REGION Network 8: SALIDAS - Baliza ROJA
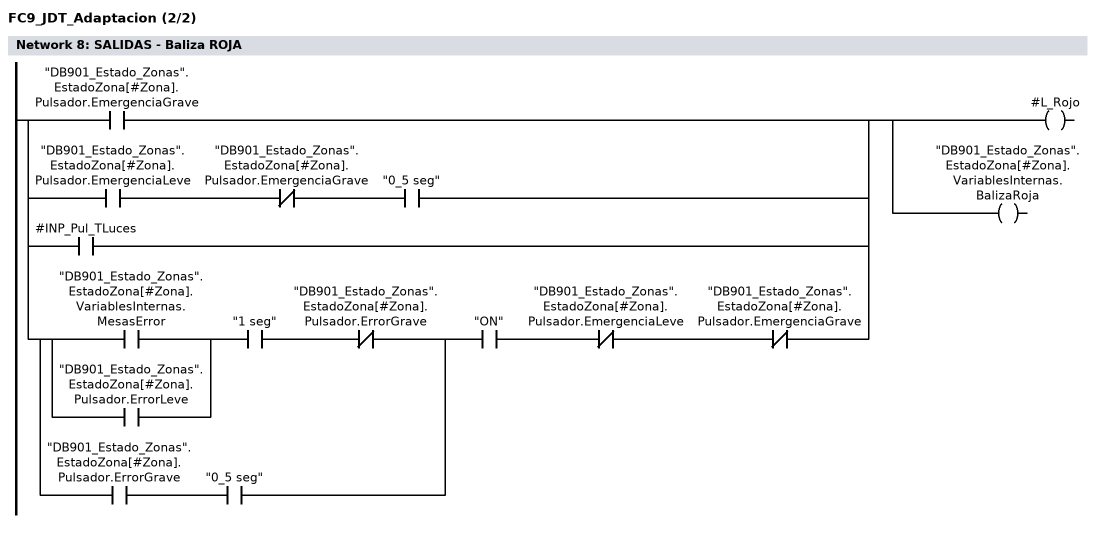
   RUNG wire#powerrail
      Contact( "DB901_Estado_Zonas".EstadoZona[#Zona].Pulsador.EmergenciaGrave )
      wire#w1
      Coil( #L_Rojo )
   END_RUNG
   RUNG wire#powerrail
      Contact( "DB901_Estado_Zonas".EstadoZona[#Zona].Pulsador.EmergenciaLeve )
      I_Contact( "DB901_Estado_Zonas".EstadoZona[#Zona].Pulsador.EmergenciaGrave )
      Contact( "0_5 seg" )
   END_RUNG wire#w1
   RUNG wire#powerrail
      Contact( #INP_Pul_TLuces )
   END_RUNG wire#w1
   RUNG wire#powerrail
      Contact( "DB901_Estado_Zonas".EstadoZona[#Zona].VariablesInternas.MesasError )
      wire#w2
      Contact( "1 seg" )
      I_Contact( "DB901_Estado_Zonas".EstadoZona[#Zona].Pulsador.ErrorGrave )
      wire#w3
      Contact( "ON" )
      I_Contact( "DB901_Estado_Zonas".EstadoZona[#Zona].Pulsador.EmergenciaLeve )
      I_Contact( "DB901_Estado_Zonas".EstadoZona[#Zona].Pulsador.EmergenciaGrave )
   END_RUNG wire#w1
   RUNG wire#powerrail
      Contact( "DB901_Estado_Zonas".EstadoZona[#Zona].Pulsador.ErrorLeve )
   END_RUNG wire#w2
   RUNG wire#powerrail
      Contact( "DB901_Estado_Zonas".EstadoZona[#Zona].Pulsador.ErrorGrave )
      Contact( "0_5 seg" )
   END_RUNG wire#w3
   RUNG wire#w1
      Coil( "DB901_Estado_Zonas".EstadoZona[#Zona].VariablesInternas.BalizaRoja )
   END_RUNG
   // the same network as SCL:
   #L_Rojo := "DB901_Estado_Zonas".EstadoZona[#Zona].Pulsador.EmergenciaGrave OR ("DB901_Estado_Zonas".EstadoZona[#Zona].Pulsador.EmergenciaLeve AND NOT "DB901_Estado_Zonas".EstadoZona[#Zona].Pulsador.EmergenciaGrave AND "0_5 seg") OR #INP_Pul_TLuces OR (((("DB901_Estado_Zonas".EstadoZona[#Zona].VariablesInternas.MesasError OR "DB901_Estado_Zonas".EstadoZona[#Zona].Pulsador.ErrorLeve) AND "1 seg" AND NOT "DB901_Estado_Zonas".EstadoZona[#Zona].Pulsador.ErrorGrave) OR ("DB901_Estado_Zonas".EstadoZona[#Zona].Pulsador.ErrorGrave AND "0_5 seg")) AND "ON" AND NOT "DB901_Estado_Zonas".EstadoZona[#Zona].Pulsador.EmergenciaLeve AND NOT "DB901_Estado_Zonas".EstadoZona[#Zona].Pulsador.EmergenciaGrave);
   "DB901_Estado_Zonas".EstadoZona[#Zona].VariablesInternas.BalizaRoja := #L_Rojo;
END_REGION
END_FUNCTION

FUNCTION_BLOCK "FB600_ControlPosicion_Quimarox"   // FB600, LAD
{ S7_Optimized_Access := 'FALSE' }
AUTHOR : Naibes
// stored: AutoNumber false, SetENOAutomatically false
   VAR_INPUT
      ID_Quimarox : UInt;
      Detector_paso_cero : Bool;
      V_Cnt_Tout_paso_Cero : UDInt;
      Dato_encoder : DInt;   // Tiene que ser una entrada del DB de encoders
   END_VAR
   VAR_OUTPUT
      numero_vagon_entrada : Int;
      avance_vagon_entrada : Int;
      avance_total : Int;
   END_VAR
   VAR
      maux_fp_detect_cero : Bool;
      mem_cnt_tout : UDInt;
      total_registros : Int;
   END_VAR
   VAR_TEMP
      contador_elementos : Int;
      pulsos_transcurridos : DInt;
      avance_vagon_ref : DInt;
      num_vag_in : Int;
      Avance_vag_inic : Int;
      aux_int : Int;
      Avance_vagon_X : Int;
      salto : Int;
      basura : Bool;
   END_VAR
BEGIN

NETWORK
TITLE = Variable provisional
//=====================================================================================================================

//=====================================================================================================================

NETWORK
TITLE = 
// Control de posicionamiento y memorias de encoder

      CALL  "FC600_ini+ref_dato_encoder_NEW"
      ( Detector_referencia := #Detector_paso_cero,
        ID_Quimarox         := #ID_Quimarox,
        dato_encoder_actual := #Dato_encoder,
        V_cnt_tout_refresco := #V_Cnt_Tout_paso_Cero,
        m_aux_pf_detect     := #maux_fp_detect_cero,
        MEM_CNT_TOUT        := #mem_cnt_tout
      );


NETWORK
TITLE = Variable provisional
      SET;
      A     "DB600_ConfigQuimarox".Quimarox[#ID_Quimarox].datos_config.DatosTrabajo.Error_Referenciacion;  // #Error_Referenciacion
      R     "DB600_ConfigQuimarox".Quimarox[#ID_Quimarox].datos_config.DatosTrabajo.Memoria_Inicializacion;  //#Mem_Inicializacion

NETWORK
TITLE = Borrado de DB Posiciones asociadas a elementos
// aqui se borran todas las posiciones asociadas a los elementos para luego 
// posteriormente cargar los datos que correspondan. Esto lo hacemos antes de 
// comprobar si está inicializado o no para que si perdemos la referencia dejemos 
// de tener datos.
//=====================================================================================================================

      L     1;  //Iniciamos Cont. Bytes a Borrar     Cuidado con los temporales, inicializar siempre
      T     #contador_elementos;


bucl: NOP   0;
//=====================================================================================================================
//limpia los datos antes de calcular los nuevos

      SET;
      R     "DB602_ElementosQuimarox".Quimarox[#ID_Quimarox].Elementos[#contador_elementos].Hay_Carrier_en_ventana;  //Vagon_en_Ventana
      L     0;
      T     "DB602_ElementosQuimarox".Quimarox[#ID_Quimarox].Elementos[#contador_elementos].Numero_carrier;  //Vagon_Asociado
      T     "DB602_ElementosQuimarox".Quimarox[#ID_Quimarox].Elementos[#contador_elementos].Avance_carrier;  //Posicion_Vagon


      L     #contador_elementos;
      L     "CTE_MaxNumElementos";
      >=I;
      JC    cont;

      L     1;
      L     #contador_elementos;
      +I;
      T     #contador_elementos;

      JU    bucl;
//=====================================================================================================================

NETWORK
TITLE = 
//=====================================================================================================================

cont: AN    "DB600_ConfigQuimarox".Quimarox[#ID_Quimarox].datos_config.DatosTrabajo.Memoria_Inicializacion;
      JC    fin1;  //el primer vagon y no podemos calcular nada

//=====================================================================================================================

NETWORK
TITLE = 
// con el dato del encoder de referencia del primer vagon calculamos el elemento 
// que se encuentra en la entrada del sorter para utilizarlo de vagon de referencia
//===================================================================================================
//aqui comprobaremos si ha pasado por el máximo o no y en funcion de eso calcularemos el numero
//de pulsos que han transcurrido desde la referenciación del primer vagon
//====================================================================================================

      L     "DB600_ConfigQuimarox".Quimarox[#ID_Quimarox].datos_config.DatosTrabajo.Memoria_Dato_Encoder;  //#Mem_Dato_Encoder
      L     #Dato_encoder;
      >D;
      JCN   MEN;

      L     "DB600_ConfigQuimarox".Quimarox[#ID_Quimarox].datos_config.maximo_encoder;
      L     "DB600_ConfigQuimarox".Quimarox[#ID_Quimarox].datos_config.DatosTrabajo.Memoria_Dato_Encoder;
      -D;
      L     #Dato_encoder;
      +D;
      T     #pulsos_transcurridos;
      JU    CLC;

//=====================================================================================================================

MEN:  L     #Dato_encoder;
      L     "DB600_ConfigQuimarox".Quimarox[#ID_Quimarox].datos_config.DatosTrabajo.Memoria_Dato_Encoder;
      -D;
      T     #pulsos_transcurridos;


//============================================================================================================================================
// NIEVES: Calculo del avance del vagón de referencia

CLC:  L     #pulsos_transcurridos;
      DTR;
      L     "DB600_ConfigQuimarox".Quimarox[#ID_Quimarox].datos_config.relacion_mm_pulso;  // #Datos_config.relacion_mm_pulso
      *R;
      RND+;
      L     "DB600_ConfigQuimarox".Quimarox[#ID_Quimarox].datos_config.dist_ini_vag_a_phs_mm;  //distancia del punto de deteccion de referencia al punto de referencia 0
      ITD;
      +D;
      T     #avance_vagon_ref;  //en mm

//=====================================================================================================================

//con el dato del avance del vagon de referencia calculamos cual es el vagon que esta en el inicio del sorter
//y cuando ha avanzado respecto del punto de referencia para con este dato calcular la posicion del resto


NETWORK
TITLE = Calculo de posicón del primer vagón
// en funcion del avance del primer vagon calculamos cual es el vagon que se 
// encuentra en el inicio del sorter y cuanto ha avanzado desde el punto de 
// referencia
//=====================================================================================================================
//si no hace bien lo del numero de vagon revisar este punto
      L     #avance_vagon_ref;
      L     "DB600_ConfigQuimarox".Quimarox[#ID_Quimarox].datos_config.Long_Vagon_mm;
      ITD;
      /D;
      L     1;
      +D;
      DTB;
      BTI;
      T     #num_vag_in;  //Calcula y guarda Vagon en posición inicial

      L     #num_vag_in;
      L     "DB600_ConfigQuimarox".Quimarox[#ID_Quimarox].datos_config.Numero_vagones;

      <=I;
      JC    p_1;

//=====================================================================================================================

      L     #num_vag_in;
      L     "DB600_ConfigQuimarox".Quimarox[#ID_Quimarox].datos_config.Numero_vagones;
      -I;
      T     #numero_vagon_entrada;
      JU    p_2;

//=====================================================================================================================
p_1:  L     #num_vag_in;
      T     #numero_vagon_entrada;

//=====================================================================================================================
p_2:  L     #avance_vagon_ref;
      L     "DB600_ConfigQuimarox".Quimarox[#ID_Quimarox].datos_config.Long_Vagon_mm;
      MOD;
      T     #avance_vagon_entrada;
      T     #Avance_vag_inic;  //Calcula y guarda avance Vagon actual en posición inicial

      L     #pulsos_transcurridos;  // Calcula el avance total desde origen
      DTR;
      L     "DB600_ConfigQuimarox".Quimarox[#ID_Quimarox].datos_config.relacion_mm_pulso;
      *R;
      RND+;
      T     #avance_total;

//=====================================================================================================================

NETWORK
TITLE = calculo posicon vagon todos elementos
// aqui vamos realizando los saltos a cada uno de los elementos, calculamos lo que 
// ha avanzado el vagon y si entra dentro de los limites establecidos para dicho 
// elemento cargamos el numero de vagon correspondiente en la posicion asociada a 
// dicho elemento
//===================================================================================================================================

      L     1;
      T     #contador_elementos;

//=====================================================================================================================
//aqui el calculo de lo que ha avanzado el vagon para dicho elemento
//NIEVES


sige: NOP   0;

//=====================================================================================================================

      L     "DB602_ElementosQuimarox".Quimarox[#ID_Quimarox].Elementos[#contador_elementos].posicion_real_elemento;  //#datos_elemento_actual.posicion_real_elemento
      TRUNC;
      L     "DB600_ConfigQuimarox".Quimarox[#ID_Quimarox].datos_config.Long_Vagon_mm;
      ITD;
      MOD;
      T     #aux_int;
      L     "DB600_ConfigQuimarox".Quimarox[#ID_Quimarox].datos_config.Long_Vagon_mm;
      L     #aux_int;
      -I;  //Avance del vagon para el elemento tratado
      L     #Avance_vag_inic;
      +I;
      L     "DB600_ConfigQuimarox".Quimarox[#ID_Quimarox].datos_config.Long_Vagon_mm;
      MOD;
      T     #Avance_vagon_X;

//=====================================================================================================================

NETWORK
TITLE = comparación de la ventana del elemento segun grado de avance
// aqui la comparacion primero con el rango inferior y luego con el rango superior
//=====================================================================================================================
      CLR;
      =     "DB602_ElementosQuimarox".Quimarox[#ID_Quimarox].Elementos[#contador_elementos].Hay_Carrier_en_ventana;  //Inicio Validación elemento en rango Ventana


      L     "DB602_ElementosQuimarox".Quimarox[#ID_Quimarox].Elementos[#contador_elementos].ventana_minima;
      L     #Avance_vagon_X;
      >I;
      JC    vent;

//=====================================================================================================================

      L     "DB602_ElementosQuimarox".Quimarox[#ID_Quimarox].Elementos[#contador_elementos].ventana_maxima;  //apunta a la posicion maxima
      L     #Avance_vagon_X;
      <I;
      JC    vent;

      SET;
      =     "DB602_ElementosQuimarox".Quimarox[#ID_Quimarox].Elementos[#contador_elementos].Hay_Carrier_en_ventana;

//=====================================================================================================================




NETWORK
TITLE = calcular el número de vagón que corresponde
// aqui si se cumple que esta entre los dos rangos, calculamos el numero de vagon 
// que corresponde y lo cargamos en la correspondiente posicion asociada
// 
// al finalizar comprobar que no estamos en el ultimo elemento, si lo estamos, 
// saltar al final, y si no lo estamos pasa al siguiente elemento y spa sige
//=====================================================================================================================
//aqui calculamos el vagon que esta en frente del elemento
// para poder hacer el redondeo tenemos que hacer todo el cálculo en real

vent: L     "DB602_ElementosQuimarox".Quimarox[#ID_Quimarox].Elementos[#contador_elementos].posicion_real_elemento;
      L     #Avance_vag_inic;
      ITD;
      DTR;
      -R;
      L     "DB600_ConfigQuimarox".Quimarox[#ID_Quimarox].datos_config.Long_Vagon_mm;
      ITD;
      DTR;
      /R;
      RND+;
      T     #salto;
      L     #num_vag_in;
      L     #salto;
      -I;
      T     #aux_int;

      L     #aux_int;
      L     1;
      <I;
      JCN   p_3;


//=====================================================================================================================
      L     #aux_int;
      L     "DB600_ConfigQuimarox".Quimarox[#ID_Quimarox].datos_config.Numero_vagones;
      +I;
      T     #aux_int;


//=====================================================================================================================
p_3:  L     #aux_int;
      L     "DB600_ConfigQuimarox".Quimarox[#ID_Quimarox].datos_config.Numero_vagones;
      >I;
      JCN   carg;

      L     #aux_int;
      L     "DB600_ConfigQuimarox".Quimarox[#ID_Quimarox].datos_config.Numero_vagones;
      -I;
      T     #aux_int;

//=====================================================================================================================
carg: L     #aux_int;
      T     "DB602_ElementosQuimarox".Quimarox[#ID_Quimarox].Elementos[#contador_elementos].Numero_carrier;

      L     #Avance_vagon_X;
      T     "DB602_ElementosQuimarox".Quimarox[#ID_Quimarox].Elementos[#contador_elementos].Avance_carrier;

//=====================================================================================================================

      L     #contador_elementos;
      L     "CTE_MaxNumElementos";
      ==I;
      JC    fin;

      L     #contador_elementos;
      L     1;
      +I;
      T     #contador_elementos;

      JU    sige;

//=====================================================================================================================

NETWORK
TITLE = 
//=====================================================================================================================
fin:  BE;


//=====================================================================================================================
fin1: L     0;
      T     #numero_vagon_entrada;
      T     #avance_vagon_entrada;


//=====================================================================================================================
END_FUNCTION_BLOCK

FUNCTION_BLOCK "FB607_SalidaMovil_Frontal_Quimarox"   // FB607, LAD
{ S7_Optimized_Access := 'FALSE' }
// stored: AutoNumber false, SetENOAutomatically false
   VAR_INPUT
      MesaDeDescarga : UInt;
      ID_Quimarox : UInt;
      ID_Elemento : UInt;
      DestinoAsociado : UInt;
      pHs_PosicionDescarga : Bool;
      pHs_Protrusion : Bool;
      En_PosicionReposo : Bool;
      Corte_PosicionReposo : Bool;
      Corte_PosicionDesCarga : Bool;
      En_PosicionDescarga : Bool;
      Permiso_DeDesCarga : Bool;
      V_Filtro_pHsPresencia : Int;
      Pto_Ajuste_1 : Int;   // en mm (paso a lenta en posicionamiento a descarga de transportador)
      Pto_Ajuste_2 : Int;   // en mm (timeout movimiento posicion descarga del transportador)
      Pto_Ajuste_3 : Int;   // en mm (paso a lenta en posicionamiento reposo del transportador)
      Pto_Ajuste_4 : Int;   // en mm (timeout movimiento posicion reposo del transportador)
   END_VAR
   VAR_OUTPUT
      NXT_DescargaActiva : Bool;
      ElevadorEnLenta : Bool;
      PararElevador : Bool;
      Ir_PosicionReposo : Bool;
      Ir_PosicionDescarga : Bool;
   END_VAR
   VAR
      FILTRO_pHsPresencia : "FB910_CNT_UHS";
      EstadoAsociadoEnMesa : UInt;
      Ultimo_PeineTratado : UInt;
      Aux_PeineEnDesCarga { ExternalAccessible := 'False'; ExternalVisible := 'False'; ExternalWritable := 'False'} : UInt;
   END_VAR
   VAR_TEMP
      MesaQuimarox : UInt;
      NumeroUT : UInt;
      Vagon_Siguiente : Int;
      EsMesaTL : Bool;
      FILTRO_PosicionDesCarga : Bool;
   END_VAR
BEGIN

NETWORK
TITLE = ERROR - Rearme
/////////////////////////////////////////////////////////////
/////////////////////////////////////////////////////////////
/////////////////////////////////////////////////////////////
// Rearne de Errores
      SET;
      A     "DB902_Estado_ZonaMesa".EstadoMesas[#MesaDeDescarga].Rearme_CBx;
      O     "DB902_Estado_ZonaMesa".EstadoMesas[#MesaDeDescarga].PerReset_CBx;
      R     "DB900_Estado_Mesas".EstadoVI[#MesaDeDescarga].Error_Mx;
      R     "DB900_Estado_Mesas".EstadoVI[#MesaDeDescarga].Err_Protusion;
      R     "DB900_Estado_Mesas".EstadoVI[#MesaDeDescarga].Err_TOut_Avance_E1_E3;
      R     "DB900_Estado_Mesas".EstadoVI[#MesaDeDescarga].Err_Tout_Sacar;
      R     "DB900_Estado_Mesas".EstadoVI[#MesaDeDescarga].Err_Tout_Recoger;

      R     "DB900_Estado_Mesas".EstadoVI[#MesaDeDescarga].Err_DatosPLC;



NETWORK
TITLE = HMI - Entradas y Salidas de la Mesa
/////////////////////////////////////////////////////////////
/////////////////////////////////////////////////////////////
/////////////////////////////////////////////////////////////
// Entradas
      SET;
      A     #pHs_PosicionDescarga;
      =     "DB904_Estado_Maquinas".EstadoVI[#MesaDeDescarga].Byte7_bit4;
      SET;
      A     #pHs_Protrusion;
      =     "DB904_Estado_Maquinas".EstadoVI[#MesaDeDescarga].Byte9_bit0;

      SET;
      A     #En_PosicionReposo;
      =     "DB904_Estado_Maquinas".EstadoVI[#MesaDeDescarga].Byte8_bit4;
      SET;
      A     #Corte_PosicionReposo;
      =     "DB904_Estado_Maquinas".EstadoVI[#MesaDeDescarga].Byte7_bit6;
      SET;
      A     #Corte_PosicionDesCarga;
      =     "DB904_Estado_Maquinas".EstadoVI[#MesaDeDescarga].Byte7_bit7;
      SET;
      A     #En_PosicionDescarga;
      =     "DB904_Estado_Maquinas".EstadoVI[#MesaDeDescarga].Byte8_bit5;


// Salidas
      SET;
      A     #NXT_DescargaActiva;
      =     "DB900_Estado_Mesas".EstadoVI[#MesaDeDescarga].Sa_Giro_180;
      SET;
      A     #Ir_PosicionReposo;
      =     "DB900_Estado_Mesas".EstadoVI[#MesaDeDescarga].Sa_Trans_Baj;
      SET;
      A     #Ir_PosicionDescarga;
      =     "DB900_Estado_Mesas".EstadoVI[#MesaDeDescarga].Sa_Trans_Sub;



NETWORK
TITLE = Comprobacion de que la MESA es de TRACKING
/////////////////////////////////////////////////////////////////////////////////////
/////////////////////////////////////////////////////////////////////////////////////
/////////////////////////////////////////////////////////////////////////////////////
// Comprobar si es una Mesa de Tracking o Routing
      SET;
      A     "DB850_DefinicionMesas".Mesa[#MesaDeDescarga].ConfigMesa.MesaTL;
      =     #EsMesaTL;



NETWORK
TITLE = Inicializacio PREVIA
/////////////////////////////////////////////////////////////////////////////////////
/////////////////////////////////////////////////////////////////////////////////////
/////////////////////////////////////////////////////////////////////////////////////
      CLR;
      =     #ElevadorEnLenta;
      =     #PararElevador;

      CLR;
      =     #NXT_DescargaActiva;

      CLR;
      =     #Ir_PosicionReposo;
      =     #Ir_PosicionDescarga;



NETWORK
TITLE = SISTEMA - Reset
/////////////////////////////////////////////////////////////
/////////////////////////////////////////////////////////////
/////////////////////////////////////////////////////////////
// - Existe RESET ??
      SET;
      AN    "DB902_Estado_ZonaMesa".EstadoMesas[#MesaDeDescarga].PerReset_CBx;  //#Estado_CBx.PerReset_CBx
      JC    NoRealizandose_Reset;

      L     0;
      T     #EstadoAsociadoEnMesa;
      T     #Ultimo_PeineTratado;


/////////////////////////////////////////////////////////////
/////////////////////////////////////////////////////////////
/////////////////////////////////////////////////////////////
// - Final Tratamiento del RESET
NoRealizandose_Reset:NOP   0;



NETWORK
TITLE = >>>>>>>>>>>>>>>>>>>>>>>>>>>>>>>>>>>>>>>>>>>>>>>>>>>>>>>>>>>>>>>>>>>

REGION Network 7: FILTRO - pHs de Presencia
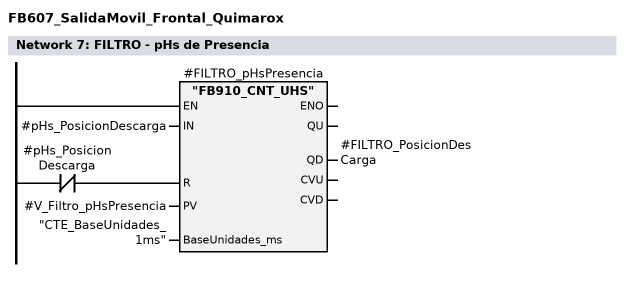
   RUNG wire#powerrail
      #FILTRO_pHsPresencia(R := wire#w1, IN := #pHs_PosicionDescarga, PV := #V_Filtro_pHsPresencia, BaseUnidades_ms := "CTE_BaseUnidades_1ms", QU =>, QD => #FILTRO_PosicionDesCarga, CVU =>, CVD =>)
   END_RUNG
   RUNG wire#powerrail
      I_Contact( #pHs_PosicionDescarga )
   END_RUNG wire#w1
   // the same network as SCL:
   #FILTRO_pHsPresencia(IN := #pHs_PosicionDescarga,   // "FB910_CNT_UHS"
                        R := NOT #pHs_PosicionDescarga,
                        PV := #V_Filtro_pHsPresencia,
                        BaseUnidades_ms := "CTE_BaseUnidades_1ms",
                        QD => #FILTRO_PosicionDesCarga);
END_REGION

NETWORK
TITLE = >>>>>>>>>>>>>>>>>>>>>>>>>>>>>>>>>>>>>>>>>>>>>>>>>>>>>>>>>>>>>>>>>>>

NETWORK
TITLE = Control Etapa activa >>> DISTRIBUCION
/////////////////////////////////////////////////////////////////////////////////////
/////////////////////////////////////////////////////////////////////////////////////
/////////////////////////////////////////////////////////////////////////////////////
// listado de saltos de programa
      L     #EstadoAsociadoEnMesa;

      JL    ETAPA_PorDefecto;
      JU    ETAPA_00_EnReset;
      JU    ETAPA_01_EnReposo;

      JU    ETAPA_02_EsperaPermisoDeDescarga;
      JU    ETAPA_03_MoverPosicionDescarga;
      JU    ETAPA_04_PreparadoParaDescarga;
      JU    ETAPA_05_FinDescarga;
      JU    ETAPA_06_MoverPosicionReposo;

      JU    ETAPA_PorDefecto;
      JU    ETAPA_PorDefecto;
      JU    ETAPA_PorDefecto;

      JU    ETAPA_10_ResetVacio_EsperaDesCargaDePeine;
      JU    ETAPA_11_ResetVacio_RecogerCargaDePeine;
      JU    ETAPA_12_ResetVacio_MoverPosicionReposo;
      JU    ETAPA_13_ResetCargado_EsperaPermisoDeDesCarga;
      JU    ETAPA_14_ResetCargado_MoverPosicionReposo;

ETAPA_PorDefecto:JU    FinFuncion;




NETWORK
TITLE = ETAPA 00 >>> En Reset
/////////////////////////////////////////////////////////////////////////////////////
/////////////////////////////////////////////////////////////////////////////////////
/////////////////////////////////////////////////////////////////////////////////////
ETAPA_00_EnReset:NOP   0;
      CLR;
      =     #Ir_PosicionReposo;
      =     #Ir_PosicionDescarga;

/////////////////////////////////////////////////////////////////////////////////////
// error de protusion
      SET;
      AN    #pHs_Protrusion;
      JC    ErrorProtrusion;

/////////////////////////////////////////////////////////////////////////////////////
// Tiene que estar en Marcha y Sin Error para continuar
      SET;
      AN    "DB902_Estado_ZonaMesa".EstadoMesas[#MesaDeDescarga].Marcha_CBx;
      O     "DB902_Estado_ZonaMesa".EstadoMesas[#MesaDeDescarga].Error_CBx;
      JC    ET00_PararElevador;


/////////////////////////////////////////////////////////////////////////////////////
// En Resposo
      SET;
      A     #En_PosicionReposo;
      JC    ET00_IrEtapa_01_EnReposo;


/////////////////////////////////////////////////////////////////////////////////////
// NO Reposo - Vacio
      SET;
      AN    #FILTRO_PosicionDesCarga;
      JC    ET00_Reset_10_ResetVacio_EsperaDesCargaDePeine;

/////////////////////////////////////////////////////////////////////////////////////
// NO Reposo - Con Carga
      SET;
      A     #FILTRO_PosicionDesCarga;
      JC    ET00_Reset_13_ResetCargado_EsperaPermisoDeDesCarga;


/////////////////////////////////////////////////////////////////////////////////////
// Final del Reparto  ?????? No DEBE LLEGAR AQUI
      BE;




/////////////////////////////////////////////////////////////////////////////////////
/////////////////////////////////////////////////////////////////////////////////////
/////////////////////////////////////////////////////////////////////////////////////
ET00_PararElevador:NOP   0;
      SET;
      =     #PararElevador;
      BE;


/////////////////////////////////////////////////////////////////////////////////////
/////////////////////////////////////////////////////////////////////////////////////
/////////////////////////////////////////////////////////////////////////////////////
ET00_IrEtapa_01_EnReposo:NOP   0;
      L     1;
      T     #EstadoAsociadoEnMesa;
      JU    ETAPA_01_EnReposo;


/////////////////////////////////////////////////////////////////////////////////////
/////////////////////////////////////////////////////////////////////////////////////
/////////////////////////////////////////////////////////////////////////////////////
ET00_Reset_10_ResetVacio_EsperaDesCargaDePeine:NOP   0;
      L     10;
      T     #EstadoAsociadoEnMesa;
      JU    ETAPA_10_ResetVacio_EsperaDesCargaDePeine;


/////////////////////////////////////////////////////////////////////////////////////
/////////////////////////////////////////////////////////////////////////////////////
/////////////////////////////////////////////////////////////////////////////////////
ET00_Reset_13_ResetCargado_EsperaPermisoDeDesCarga:NOP   0;
      L     13;
      T     #EstadoAsociadoEnMesa;
      JU    ETAPA_13_ResetCargado_EsperaPermisoDeDesCarga;



NETWORK
TITLE = ETAPA 01 >>> En Reposo
/////////////////////////////////////////////////////////////////////////////////////
/////////////////////////////////////////////////////////////////////////////////////
/////////////////////////////////////////////////////////////////////////////////////
// Estado de reposo esperando a que llegue una carga para este destino
ETAPA_01_EnReposo:NOP   0;
      SET;
      AN    #En_PosicionReposo;
      JC    ET01_IrEtapa_14_MoverPosicionReposo;

/////////////////////////////////////////////////////////////////////////////////////
// miramos si ya hemos comprobado el peine que está delante nuestro
      SET;
      L     "DB602_ElementosQuimarox".Quimarox[#ID_Quimarox].Elementos[#ID_Elemento].Numero_carrier;
      L     #Ultimo_PeineTratado;
      ==I;
      JC    ET01_SinPeineEnVentana;

/////////////////////////////////////////////////////////////////////////////////////
// si no hemos comprobado el peine, comprobamos si tenemos un peine en ventana
      SET;
      AN    "DB602_ElementosQuimarox".Quimarox[#ID_Quimarox].Elementos[#ID_Elemento].Hay_Carrier_en_ventana;
      JC    ET01_SinPeineEnVentana;

/////////////////////////////////////////////////////////////////////////////////////
// si no ha saltado es porque el carrier está en ventana. Comprobamos si es para nosotros
      L     "DB602_ElementosQuimarox".Quimarox[#ID_Quimarox].Elementos[#ID_Elemento].Numero_carrier;
      T     #Aux_PeineEnDesCarga;

      SET;
      L     "DB601_PeinesQuimarox".Quimarox[#ID_Quimarox].vagon[#Aux_PeineEnDesCarga].Destino_principal;
      L     #DestinoAsociado;
      ==I;
      JC    ET01_PeineParaLaMesa;

/////////////////////////////////////////////////////////////////////////////////////
// si no es para mi, me guardo que he chequeado el peine para no volver a comprobarlo
      L     "DB602_ElementosQuimarox".Quimarox[#ID_Quimarox].Elementos[#ID_Elemento].Numero_carrier;
      T     #Ultimo_PeineTratado;
      BE;


/////////////////////////////////////////////////////////////////////////////////////
/////////////////////////////////////////////////////////////////////////////////////
/////////////////////////////////////////////////////////////////////////////////////
ET01_SinPeineEnVentana:NOP   0;
      SET;  // Esta TOTALMENTE libre ?
      A(;
      O     #FILTRO_PosicionDesCarga;
      ON    #pHs_Protrusion;
      );
      JCN   FinFuncion;
      JU    ErrorProtrusion;


/////////////////////////////////////////////////////////////////////////////////////
/////////////////////////////////////////////////////////////////////////////////////
/////////////////////////////////////////////////////////////////////////////////////
ET01_PeineParaLaMesa:NOP   0;
      L     2;
      T     #EstadoAsociadoEnMesa;
      L     "DB602_ElementosQuimarox".Quimarox[#ID_Quimarox].Elementos[#ID_Elemento].Numero_carrier;
      T     #Ultimo_PeineTratado;

      JU    ETAPA_02_EsperaPermisoDeDescarga;


/////////////////////////////////////////////////////////////////////////////////////
/////////////////////////////////////////////////////////////////////////////////////
/////////////////////////////////////////////////////////////////////////////////////
ET01_IrEtapa_14_MoverPosicionReposo:NOP   0;
      L     14;
      T     #EstadoAsociadoEnMesa;
      JU    ETAPA_14_ResetCargado_MoverPosicionReposo;


NETWORK
TITLE = ETAPA 02 >>> Etapa Espera de Permiso de Descarga
/////////////////////////////////////////////////////////////////////////////////////
/////////////////////////////////////////////////////////////////////////////////////
/////////////////////////////////////////////////////////////////////////////////////
// Espera a Permiso de Descarga. Antes de iniciar el Ciclo de Descarga
ETAPA_02_EsperaPermisoDeDescarga:NOP   0;
      SET;
      A     #Permiso_DeDesCarga;
      JC    ET02_IrEtapa_03_MoverPosicionDesCarga;

      SET;  // No se puede Iniciar el Ciclo
      =     #PararElevador;
      BE;

/////////////////////////////////////////////////////////////////////////////////////
// Esta el Permiso de Descarga >>> Activar Ciclo de Descarga
ET02_IrEtapa_03_MoverPosicionDesCarga:NOP   0;
      L     3;
      T     #EstadoAsociadoEnMesa;

      JU    ETAPA_03_MoverPosicionDescarga;



NETWORK
TITLE = ETAPA 03 >>> Mover a Posicion de Descarga
/////////////////////////////////////////////////////////////////////////////////////
/////////////////////////////////////////////////////////////////////////////////////
/////////////////////////////////////////////////////////////////////////////////////
// inicio del proceso de descarga
// antes de iniciar la descarga tenemos que colocar el transportador en la posicion de descarga
ETAPA_03_MoverPosicionDescarga:NOP   0;
      SET;
      A     #En_PosicionDescarga;
      JC    ET03_IrEtapa_04_PreparadoParaDesCarga;

/////////////////////////////////////////////////////////////////////////////////////
      SET;
      =     #Ir_PosicionDescarga;
      CLR;
      =     #Ir_PosicionReposo;

/////////////////////////////////////////////////////////////////////////////////////
// como estamos metiendo el transportador, tenemos que vigilar que no tarda demasiado en entrar
      L     "DB602_ElementosQuimarox".Quimarox[#ID_Quimarox].Elementos[#ID_Elemento].Avance_carrier;  // #datos_elemento.Avance_carrier
      L     #Pto_Ajuste_1;
      <=I;
      JC    ET03_VelocidadNormal;

      SET;
      =     #ElevadorEnLenta;

      L     "DB602_ElementosQuimarox".Quimarox[#ID_Quimarox].Elementos[#ID_Elemento].Avance_carrier;  //#datos_elemento.Avance_carrier
      L     #Pto_Ajuste_2;
      >=I;
      JC    ErrorMoverPosicionDescarga;  // error de movimiento al sacar el transportador

      BE;


/////////////////////////////////////////////////////////////////////////////////////
ET03_VelocidadNormal:CLR;
      =     #ElevadorEnLenta;
      BE;

/////////////////////////////////////////////////////////////////////////////////////
ET03_IrEtapa_04_PreparadoParaDesCarga:CLR;
      =     #Ir_PosicionDescarga;
      L     4;
      T     #EstadoAsociadoEnMesa;

      JU    ETAPA_04_PreparadoParaDescarga;



NETWORK
TITLE = ETAPA 04 >>> Etapa Preparado para el Proceso de Descarga
/////////////////////////////////////////////////////////////////////////////////////
/////////////////////////////////////////////////////////////////////////////////////
/////////////////////////////////////////////////////////////////////////////////////
// espera a la descarga activa
// antes de iniciar la descarga tenemos que esperar a ver el detector de la descarga
ETAPA_04_PreparadoParaDescarga:NOP   0;
      SET;
      =     #NXT_DescargaActiva;

      SET;
      A     #FILTRO_PosicionDesCarga;
      A     #pHs_Protrusion;
      JC    ET04_IrEtapa_05_FinDescarga;


/////////////////////////////////////////////////////////////////////////////////////
// tenemos que comprobar si seguimos en la ventana, sino nos retiramos
      SET;
      AN    #pHs_Protrusion;
      JC    ErrorProtrusion;

/////////////////////////////////////////////////////////////////////////////////////
      SET;
      A     "DB602_ElementosQuimarox".Quimarox[#ID_Quimarox].Elementos[#ID_Elemento].Hay_Carrier_en_ventana;
      JC    FinFuncion;


/////////////////////////////////////////////////////////////////////////////////////
      SET;
      AN    "DB602_ElementosQuimarox".Quimarox[#ID_Quimarox].Elementos[#ID_Elemento].Hay_Carrier_en_ventana;
      JC    ET04_IrEtapa_06_MoverPosicionReposo;

      BE;


/////////////////////////////////////////////////////////////////////////////////////
ET04_IrEtapa_06_MoverPosicionReposo:NOP   0;
      L     6;
      T     #EstadoAsociadoEnMesa;
      JU    ETAPA_06_MoverPosicionReposo;

/////////////////////////////////////////////////////////////////////////////////////
// si hemos visto el detector, es que nos tenemos que poner en el estado de descarga activa.
ET04_IrEtapa_05_FinDescarga:NOP   0;
      L     5;
      T     #EstadoAsociadoEnMesa;
      JU    ETAPA_05_FinDescarga;



NETWORK
TITLE = ETAPA 05 >>> Fin Descarga
/////////////////////////////////////////////////////////////////////////////////////
/////////////////////////////////////////////////////////////////////////////////////
/////////////////////////////////////////////////////////////////////////////////////
// antes de saltar al inicio proceso reposo, vamos a ver si el siguiente peine que va a llegar
// tiene también una carga para nosotros. Para eso tenemos que sacar el dato del peine siguiente.
ETAPA_05_FinDescarga:NOP   0;
      SET;
      =     #NXT_DescargaActiva;

/////////////////////////////////////////////////////////////////////////////////////
/////////////////////////////////////////////////////////////////////////////////////
/////////////////////////////////////////////////////////////////////////////////////
// COMPROBAR EL TIPO DE MESA
      L     "CTE_Evento_QDES";
      T     "DB601_PeinesQuimarox".Quimarox[#ID_Quimarox].vagon[#Aux_PeineEnDesCarga].EventoAGenerar;
      L     #MesaDeDescarga;
      L     "CTE_OffsetMesa";
      +I;
      T     "DB601_PeinesQuimarox".Quimarox[#ID_Quimarox].vagon[#Aux_PeineEnDesCarga].Mesa_descarga;

      SET;
      AN    #EsMesaTL;
      JC    TRACKING_PasoDeDatos;
      JU    ROUTING_PasoDeDatos;

/////////////////////////////////////////////////////////////////////////////////////
// MESA DE ROUTING
ROUTING_PasoDeDatos:NOP   0;
      JU    FINAL_PasoDeDatos;

/////////////////////////////////////////////////////////////////////////////////////
// MESA DE TRACKING
// ANTES DE CREAR LA UT, TENGO QUE COMPROBAR SI EL MCKEY ES 0
TRACKING_PasoDeDatos:NOP   0;
      SET;
      L     "DB601_PeinesQuimarox".Quimarox[#ID_Quimarox].vagon[#Aux_PeineEnDesCarga].DatosCarga.Mckey;
      L     0;
      ==D;
      JC    TRACKING_CrearNueva_UT;

/////////////////////////////////////////////////////////////////////////////////////
// AQUI GENERAMOS LA UT EN LA MESA DE DESTINO CON MCKEY CONOCIDO
      CALL  "FC721_CrearUT_EnMesa"
      ( McKey      := "DB601_PeinesQuimarox".Quimarox[#ID_Quimarox].vagon[#Aux_PeineEnDesCarga].DatosCarga.Mckey,
        MesaActual := #MesaDeDescarga,
        NumeroUT   := #NumeroUT
      );

      L     11;  // Cambio de Mesa de la UT
      T     "DB812_UTs_Control".UT[#NumeroUT].EstadoEmisionUT;

      L     "DB601_PeinesQuimarox".Quimarox[#ID_Quimarox].vagon[#Aux_PeineEnDesCarga].DatosCarga.MesaDestino;
      T     "DB812_UTs_Control".UT[#NumeroUT].MesaDestino;
      T     "DB813_UTs_Ruta".UT[#NumeroUT].Ruta[0];

      JU    FINAL_PasoDeDatos;

/////////////////////////////////////////////////////////////////////////////////////
// AQUI GENERAMOS LA UT EN LA MESA DE DESTINO CON MCKEY DESCONOCIDO
TRACKING_CrearNueva_UT:NOP   0;
      CALL  "FC723_InsertarUT_EnMesa"
      ( MesaActual := #MesaDeDescarga,
        NumeroUT   := #NumeroUT
      );

      L     12;  // Aviso de Nueva UT en la Mesa
      T     "DB812_UTs_Control".UT[#NumeroUT].EstadoEmisionUT;

      JU    FINAL_PasoDeDatos;


/////////////////////////////////////////////////////////////////////////////////////
/////////////////////////////////////////////////////////////////////////////////////
/////////////////////////////////////////////////////////////////////////////////////
FINAL_PasoDeDatos:NOP   0;
      L     6;
      T     #EstadoAsociadoEnMesa;
      JU    ETAPA_06_MoverPosicionReposo;



NETWORK
TITLE = ETAPA 06 >>> Mover a Posicion de Reposo
/////////////////////////////////////////////////////////////////////////////////////
/////////////////////////////////////////////////////////////////////////////////////
/////////////////////////////////////////////////////////////////////////////////////
// inicio del proceso de vuelta a reposo
ETAPA_06_MoverPosicionReposo:NOP   0;
      CLR;
      =     #NXT_DescargaActiva;

      SET;
      A     #En_PosicionReposo;
      JC    ET06_REPOSO_IrEtapa_01_EnReposo;

/////////////////////////////////////////////////////////////////////////////////////
      SET;
      =     #Ir_PosicionReposo;

      L     "DB602_ElementosQuimarox".Quimarox[#ID_Quimarox].Elementos[#ID_Elemento].Avance_carrier;  //#datos_elemento.Avance_carrier
      L     #Pto_Ajuste_3;
      <=I;
      JC    ET06_REPOSO_VelocidadNormal;

      SET;
      =     #ElevadorEnLenta;

/////////////////////////////////////////////////////////////////////////////////////
      SET;
      L     "DB602_ElementosQuimarox".Quimarox[#ID_Quimarox].Elementos[#ID_Elemento].Avance_carrier;  // #datos_elemento.Avance_carrier
      L     #Pto_Ajuste_4;
      >=I;
      JC    ErrorMoverPosicionReposo;  // error de movimiento al meter el transportador

/////////////////////////////////////////////////////////////////////////////////////
      SET;
      AN    "DB602_ElementosQuimarox".Quimarox[#ID_Quimarox].Elementos[#ID_Elemento].Hay_Carrier_en_ventana;  //#datos_elemento.Hay_Carrier_en_ventana
      JC    ErrorMoverPosicionReposo;

      BE;

/////////////////////////////////////////////////////////////////////////////////////
ET06_REPOSO_VelocidadNormal:NOP   0;
      CLR;
      =     #ElevadorEnLenta;
      BE;

/////////////////////////////////////////////////////////////////////////////////////
ET06_REPOSO_IrEtapa_01_EnReposo:NOP   0;
      CLR;
      =     #Ir_PosicionReposo;
      =     #ElevadorEnLenta;

      L     1;
      T     #EstadoAsociadoEnMesa;
      BE;



NETWORK
TITLE = >>>>>>>>>>>>>>>>>>>>>>>>>>>>>>>>>>>>>>>>>>>>>>>>>>>>>>>>>>>>>>>>>>>

NETWORK
TITLE = ETAPA 10 >>> RESET VACIO - EsperaDesCarga del Peine
/////////////////////////////////////////////////////////////////////////////////////
/////////////////////////////////////////////////////////////////////////////////////
/////////////////////////////////////////////////////////////////////////////////////
// Mirar si el peine Actal Existe Carga para el elemento
ETAPA_10_ResetVacio_EsperaDesCargaDePeine:NOP   0;
      SET;
      =     #PararElevador;


/////////////////////////////////////////////////////////////////////////////////////
// error de protusion
      SET;
      AN    #pHs_Protrusion;
      JC    ErrorProtrusion;

/////////////////////////////////////////////////////////////////////////////////////
// si no hemos comprobado el peine, comprobamos si tenemos un peine en ventana
      SET;
      AN    "DB602_ElementosQuimarox".Quimarox[#ID_Quimarox].Elementos[#ID_Elemento].Hay_Carrier_en_ventana;
      JC    ET10_RESET_IrEtapa_12_MoverPosicionReposo;

/////////////////////////////////////////////////////////////////////////////////////
// Comprobamos si es para nosotros, El peine
      L     "DB602_ElementosQuimarox".Quimarox[#ID_Quimarox].Elementos[#ID_Elemento].Numero_carrier;
      T     #Aux_PeineEnDesCarga;

      SET;
      L     "DB601_PeinesQuimarox".Quimarox[#ID_Quimarox].vagon[#Aux_PeineEnDesCarga].Destino_principal;
      L     #DestinoAsociado;
      ==I;
      JC    ET10_RESET_IrEtapa_11_RecogerCargaDePeine;

/////////////////////////////////////////////////////////////////////////////////////
// si no es para mi, me guardo que he chequeado el peine para no volver a comprobarlo
      L     "DB602_ElementosQuimarox".Quimarox[#ID_Quimarox].Elementos[#ID_Elemento].Numero_carrier;
      T     #Ultimo_PeineTratado;

      JU    ET10_RESET_IrEtapa_12_MoverPosicionReposo;


/////////////////////////////////////////////////////////////////////////////////////
/////////////////////////////////////////////////////////////////////////////////////
/////////////////////////////////////////////////////////////////////////////////////
ET10_RESET_IrEtapa_11_RecogerCargaDePeine:NOP   0;

      L     "DB602_ElementosQuimarox".Quimarox[#ID_Quimarox].Elementos[#ID_Elemento].Numero_carrier;
      T     #Ultimo_PeineTratado;

      L     11;
      T     #EstadoAsociadoEnMesa;
      JU    ETAPA_11_ResetVacio_RecogerCargaDePeine;

/////////////////////////////////////////////////////////////////////////////////////
/////////////////////////////////////////////////////////////////////////////////////
/////////////////////////////////////////////////////////////////////////////////////
ET10_RESET_IrEtapa_12_MoverPosicionReposo:NOP   0;
      L     "DB602_ElementosQuimarox".Quimarox[#ID_Quimarox].Elementos[#ID_Elemento].Numero_carrier;
      T     #Ultimo_PeineTratado;

      L     12;
      T     #EstadoAsociadoEnMesa;
      JU    ETAPA_12_ResetVacio_MoverPosicionReposo;



NETWORK
TITLE = ETAPA 11 >>> RESET VACIO - Recoger Carga Del Peine
/////////////////////////////////////////////////////////////////////////////////////
/////////////////////////////////////////////////////////////////////////////////////
/////////////////////////////////////////////////////////////////////////////////////
// Recoger la Carga a Velocidad Lenta por SEGURIDAD
// Deberia descargar SIEMPE >>> SINO NO PASAR AQUI
ETAPA_11_ResetVacio_RecogerCargaDePeine:NOP   0;
      SET;
      =     #ElevadorEnLenta;

/////////////////////////////////////////////////////////////////////////////////////
      SET;
      AN    #Permiso_DeDesCarga;
      JC    ET11_PararElevador;


/////////////////////////////////////////////////////////////////////////////////////
      SET;
      =     #NXT_DescargaActiva;

      SET;
      A     #FILTRO_PosicionDesCarga;
      A     #pHs_Protrusion;
      JC    ET11_IrEtapa_5_FinDescarga;


/////////////////////////////////////////////////////////////////////////////////////
// Error de Carga
      SET;
      AN    #pHs_Protrusion;
      JC    ErrorProtrusion;

/////////////////////////////////////////////////////////////////////////////////////
// Si no esta en VENTADA --- ERROR
      SET;
      AN    "DB602_ElementosQuimarox".Quimarox[#ID_Quimarox].Elementos[#ID_Elemento].Hay_Carrier_en_ventana;
      JC    ErrorDatosCargada;

      BE;

/////////////////////////////////////////////////////////////////////////////////////
/////////////////////////////////////////////////////////////////////////////////////
/////////////////////////////////////////////////////////////////////////////////////
ET11_PararElevador:NOP   0;
      SET;
      =     #PararElevador;
      BE;


/////////////////////////////////////////////////////////////////////////////////////
/////////////////////////////////////////////////////////////////////////////////////
/////////////////////////////////////////////////////////////////////////////////////
// si hemos visto el detector, es que nos tenemos que poner en el estado de descarga activa.
ET11_IrEtapa_5_FinDescarga:NOP   0;
      L     5;
      T     #EstadoAsociadoEnMesa;
      JU    ETAPA_05_FinDescarga;




NETWORK
TITLE = ETAPA 12 >>> RESET VACIO - Mover Posicion Reposo
/////////////////////////////////////////////////////////////////////////////////////
/////////////////////////////////////////////////////////////////////////////////////
/////////////////////////////////////////////////////////////////////////////////////
// Mover a Posicion Reposo >>> NO ESPERA CARGA
ETAPA_12_ResetVacio_MoverPosicionReposo:NOP   0;
      SET;
      =     #Ir_PosicionReposo;
      =     #PararElevador;


/////////////////////////////////////////////////////////////////////////////////////
      SET;
      A     #En_PosicionReposo;
      JC    ET12_RESET_IrEtapa_01_EnReposo;

      BE;


/////////////////////////////////////////////////////////////////////////////////////
/////////////////////////////////////////////////////////////////////////////////////
/////////////////////////////////////////////////////////////////////////////////////
ET12_RESET_IrEtapa_01_EnReposo:NOP   0;
      CLR;
      =     #Ir_PosicionReposo;
      =     #PararElevador;

      L     1;
      T     #EstadoAsociadoEnMesa;
      JU    ETAPA_01_EnReposo;



NETWORK
TITLE = >>>>>>>>>>>>>>>>>>>>>>>>>>>>>>>>>>>>>>>>>>>>>>>>>>>>>>>>>>>>>>>>>>>

NETWORK
TITLE = ETAPA 13 >>> RESET CARGADO - Espera De Permiso De DesCarga
/////////////////////////////////////////////////////////////////////////////////////
/////////////////////////////////////////////////////////////////////////////////////
/////////////////////////////////////////////////////////////////////////////////////
// Espera a Permiso de Descarga.
ETAPA_13_ResetCargado_EsperaPermisoDeDesCarga:NOP   0;
      SET;
      =     #NXT_DescargaActiva;
      =     #PararElevador;

/////////////////////////////////////////////////////////////////////////////////////
      SET;
      A     #Permiso_DeDesCarga;
      JC    ET13_RESET_IrEtapa_14_MoverPosicionReposo;

      BE;


/////////////////////////////////////////////////////////////////////////////////////
/////////////////////////////////////////////////////////////////////////////////////
/////////////////////////////////////////////////////////////////////////////////////
// Esta el Permiso de Descarga
ET13_RESET_IrEtapa_14_MoverPosicionReposo:NOP   0;
      L     14;
      T     #EstadoAsociadoEnMesa;
      JU    ETAPA_14_ResetCargado_MoverPosicionReposo;



NETWORK
TITLE = ETAPA 14 >>> RESET CARGADO - Mover a Posicion de Reposo
/////////////////////////////////////////////////////////////////////////////////////
/////////////////////////////////////////////////////////////////////////////////////
/////////////////////////////////////////////////////////////////////////////////////
//
ETAPA_14_ResetCargado_MoverPosicionReposo:NOP   0;
      SET;
      =     #Ir_PosicionReposo;
      =     #PararElevador;

/////////////////////////////////////////////////////////////////////////////////////
      SET;
      A     #En_PosicionReposo;
      JC    ET14_RESET_IrEtapa_01_EnReposo;

      BE;


/////////////////////////////////////////////////////////////////////////////////////
/////////////////////////////////////////////////////////////////////////////////////
/////////////////////////////////////////////////////////////////////////////////////
ET14_RESET_IrEtapa_01_EnReposo:NOP   0;
      CLR;
      =     #Ir_PosicionReposo;
      =     #PararElevador;

      L     1;
      T     #EstadoAsociadoEnMesa;
      JU    ETAPA_01_EnReposo;



NETWORK
TITLE = >>>>>>>>>>>>>>>>>>>>>>>>>>>>>>>>>>>>>>>>>>>>>>>>>>>>>>>>>>>>>>>>>>>

NETWORK
TITLE = ERRRORES DE LA MESA >>> Activacion
/////////////////////////////////////////////////////////////////////////////////////
/////////////////////////////////////////////////////////////////////////////////////
/////////////////////////////////////////////////////////////////////////////////////
ErrorProtrusion:SET;
      =     #PararElevador;
      =     "DB900_Estado_Mesas".EstadoVI[#MesaDeDescarga].Error_Mx;
      =     "DB900_Estado_Mesas".EstadoVI[#MesaDeDescarga].Err_Protusion;
      BE;

/////////////////////////////////////////////////////////////////////////////////////
/////////////////////////////////////////////////////////////////////////////////////
/////////////////////////////////////////////////////////////////////////////////////
ErrorMoverPosicionDescarga:SET;
      =     #PararElevador;
      =     "DB900_Estado_Mesas".EstadoVI[#MesaDeDescarga].Error_Mx;
      =     "DB900_Estado_Mesas".EstadoVI[#MesaDeDescarga].Err_Tout_Sacar;
      BE;

/////////////////////////////////////////////////////////////////////////////////////
/////////////////////////////////////////////////////////////////////////////////////
/////////////////////////////////////////////////////////////////////////////////////
ErrorMoverPosicionReposo:SET;
      =     #PararElevador;
      =     "DB900_Estado_Mesas".EstadoVI[#MesaDeDescarga].Error_Mx;
      =     "DB900_Estado_Mesas".EstadoVI[#MesaDeDescarga].Err_Tout_Recoger;
      BE;

/////////////////////////////////////////////////////////////////////////////////////
/////////////////////////////////////////////////////////////////////////////////////
/////////////////////////////////////////////////////////////////////////////////////
ErrorDatosCargada:NOP   0;  // error en la carga
      SET;
      =     "DB900_Estado_Mesas".EstadoVI[#MesaDeDescarga].Error_Mx;
      =     "DB900_Estado_Mesas".EstadoVI[#MesaDeDescarga].Err_DatosPLC;
      =     #PararElevador;
      BE;



NETWORK
TITLE = FIN DE LA FUNCION
/////////////////////////////////////////////////////////////////////////////////////
/////////////////////////////////////////////////////////////////////////////////////
/////////////////////////////////////////////////////////////////////////////////////
FinFuncion:BE;


END_FUNCTION_BLOCK

FUNCTION "FC602_ReservaPeine" : Void   // FC602, LAD
{ S7_Optimized_Access := 'TRUE' }
// stored: AutoNumber false, SetENOAutomatically false
   VAR_INPUT
      ID_Quimarox : UInt;
      ID_ElementoPeticion : UInt;
      TipoDeElemento : UInt;
   END_VAR
   VAR_OUTPUT
      NumeroPeineReservado : UInt;
   END_VAR
   VAR_TEMP
      PeineParaReserva : UInt;
      MesaFija : Bool;
      MesaMovilLateral : Bool;
      MesaMovilFrontal : Bool;
   END_VAR
BEGIN

NETWORK
TITLE = Inicializacion
/////////////////////////////////////////////////////////////////////////////////////
/////////////////////////////////////////////////////////////////////////////////////
/////////////////////////////////////////////////////////////////////////////////////
// Inicialización
      L     0;
      T     #NumeroPeineReservado;


/////////////////////////////////////////////////////////////////////////////////////
/////////////////////////////////////////////////////////////////////////////////////
/////////////////////////////////////////////////////////////////////////////////////
// Tipo de Mesa
      SET;  // Mesa Fija (1)
      L     #TipoDeElemento;
      L     1;
      ==I;
      S     #MesaFija;

      SET;  // Mesa Movil Lateral Fija (2)
      L     #TipoDeElemento;
      L     2;
      ==I;
      S     #MesaMovilLateral;


      SET;  // Mesa Movil Frontal (3)
      L     #TipoDeElemento;
      L     3;
      ==I;
      S     #MesaMovilFrontal;



NETWORK
TITLE = FASE 1 >>> Inicio de la Reserva
/////////////////////////////////////////////////////////////////////////////////////
/////////////////////////////////////////////////////////////////////////////////////
/////////////////////////////////////////////////////////////////////////////////////
// Primero miramos si hay un número de vagón valido.
// Si está a cero es que no se está ejecutando el control de posicion y no se puede reservar
      SET;
      A(;
      L     "DB602_ElementosQuimarox".Quimarox[#ID_Quimarox].Elementos[#ID_ElementoPeticion].Numero_carrier;
      L     0;  // #DatosElemento.ventana_minima
      ==I;
      );
      JC    EsperaParaReservar;


/////////////////////////////////////////////////////////////////////////////////////
/////////////////////////////////////////////////////////////////////////////////////
/////////////////////////////////////////////////////////////////////////////////////
// Miramos si el que tenemos delante >>> Aún no ha entrado en ventana , lo podríamos utilizar
      L     "DB602_ElementosQuimarox".Quimarox[#ID_Quimarox].Elementos[#ID_ElementoPeticion].Numero_carrier;
      T     #PeineParaReserva;

      SET;
      AN    "DB602_ElementosQuimarox".Quimarox[#ID_Quimarox].Elementos[#ID_ElementoPeticion].Hay_Carrier_en_ventana;
      A(;
      L     "DB602_ElementosQuimarox".Quimarox[#ID_Quimarox].Elementos[#ID_ElementoPeticion].Avance_carrier;
      L     "DB602_ElementosQuimarox".Quimarox[#ID_Quimarox].Elementos[#ID_ElementoPeticion].ventana_minima;
      <I;
      );
      JCN   FASE01_SiguientePeine;
      JU    ComprobarPeine_ParaReservar;


/////////////////////////////////////////////////////////////////////////////////////
/////////////////////////////////////////////////////////////////////////////////////
/////////////////////////////////////////////////////////////////////////////////////
/// Control de Numero de Peines
FASE01_SiguientePeine:NOP   0;
      L     "DB602_ElementosQuimarox".Quimarox[#ID_Quimarox].Elementos[#ID_ElementoPeticion].Numero_carrier;
      L     1;
      +I;
      T     #PeineParaReserva;

// comprobamos que no hemos superado el máximo de peines configurado
      SET;
      L     #PeineParaReserva;
      L     "DB600_ConfigQuimarox".Quimarox[#ID_Quimarox].datos_config.Numero_vagones;
      <=I;
      JC    ComprobarPeine_ParaReservar;

// si no hemos saltado, es que hemos superado el máximo, y tenemos que volver al peine 1
      L     1;
      T     #PeineParaReserva;
      JU    ComprobarPeine_ParaReservar;



NETWORK
TITLE = FASE 2 >>> Bucle de la Busqueda de la Reserva

/////////////////////////////////////////////////////////////////////////////////////
/////////////////////////////////////////////////////////////////////////////////////
/////////////////////////////////////////////////////////////////////////////////////
// Pasamos a comprobar el estado del carrier (vacio, habilitado, etc) para gestionar la reserva
ComprobarPeine_ParaReservar:NOP   0;



/////////////////////////////////////////////////////////////////////////////////////
/////////////////////////////////////////////////////////////////////////////////////
/////////////////////////////////////////////////////////////////////////////////////
// --- Vacio Totalmente >> NO Cargado y No Reservado
      SET;
      AN    "DB601_PeinesQuimarox".Quimarox[#ID_Quimarox].vagon[#PeineParaReserva].Carrier_Cargado;
      AN    "DB601_PeinesQuimarox".Quimarox[#ID_Quimarox].vagon[#PeineParaReserva].vagon_reservado_carga;

      AN    "DB601_PeinesQuimarox".Quimarox[#ID_Quimarox].vagon[#PeineParaReserva].vagon_cargado_SinDestino;
      AN    "DB601_PeinesQuimarox".Quimarox[#ID_Quimarox].vagon[#PeineParaReserva].carrier_no_utilizable;
      AN    "DB601_PeinesQuimarox".Quimarox[#ID_Quimarox].vagon[#PeineParaReserva].carrier_multiple;
      JC    GestionaReserva_PeineEncontrado;

// --- ESTA Cargado, pero NO Reservado >>> Para Mesa Fija
      SET;
      A     #MesaFija;
      A     "DB601_PeinesQuimarox".Quimarox[#ID_Quimarox].vagon[#PeineParaReserva].Carrier_Cargado;
      AN    "DB601_PeinesQuimarox".Quimarox[#ID_Quimarox].vagon[#PeineParaReserva].vagon_reservado_carga;

      AN    "DB601_PeinesQuimarox".Quimarox[#ID_Quimarox].vagon[#PeineParaReserva].vagon_cargado_SinDestino;
      AN    "DB601_PeinesQuimarox".Quimarox[#ID_Quimarox].vagon[#PeineParaReserva].carrier_no_utilizable;
      AN    "DB601_PeinesQuimarox".Quimarox[#ID_Quimarox].vagon[#PeineParaReserva].carrier_multiple;
      JC    GestionaReserva_PeineEncontrado;

// --- SI llega aqui, significa que el peine no se puede reservar, y tenemos que buscar en el siguiente
      JU    FASE02_BuscarSiguientePeine;


/////////////////////////////////////////////////////////////////////////////////////
/////////////////////////////////////////////////////////////////////////////////////
/////////////////////////////////////////////////////////////////////////////////////
// ese carrier no puede ser reservado y tenemos que mirar en el siguiente
FASE02_BuscarSiguientePeine:NOP   0;
      L     #PeineParaReserva;
      L     1;
      +I;
      T     #PeineParaReserva;

// comprobamos que no supera los límites
      SET;
      L     #PeineParaReserva;
      L     "DB600_ConfigQuimarox".Quimarox[#ID_Quimarox].datos_config.Numero_vagones;
      >I;
      JC    FASE02_SuperaMaximo_Peines;
      JU    FASE02_Continuar_BusquedaPeine;


/////////////////////////////////////////////////////////////////////////////////////
/////////////////////////////////////////////////////////////////////////////////////
/////////////////////////////////////////////////////////////////////////////////////
FASE02_SuperaMaximo_Peines:SET;
      L     1;
      T     #PeineParaReserva;
      JU    FASE02_Continuar_BusquedaPeine;


/////////////////////////////////////////////////////////////////////////////////////
/////////////////////////////////////////////////////////////////////////////////////
/////////////////////////////////////////////////////////////////////////////////////
// comprobamos que no hemos recorrido todos los peines intentando hacer una reserva sin exito
FASE02_Continuar_BusquedaPeine:NOP   0;
      SET;
      L     #PeineParaReserva;
      L     "DB602_ElementosQuimarox".Quimarox[#ID_Quimarox].Elementos[#ID_ElementoPeticion].Numero_carrier;
      ==I;
      JC    EsperaParaReservar;

// si no ha saltado es que tenemos que comprobar el siguiente carrier
      JU    ComprobarPeine_ParaReservar;



NETWORK
TITLE = FASE FINAL >>> Peine Encontrado >>> Activar Reserva
/////////////////////////////////////////////////////////////////////////////////////
/////////////////////////////////////////////////////////////////////////////////////
/////////////////////////////////////////////////////////////////////////////////////
// gestionamos la reserva
GestionaReserva_PeineEncontrado:NOP   0;
//      BE                         // PRUEBAS DE RESERVA CUIDADO!!!!

      SET;  // activamos el bit de reservado
      =     "DB601_PeinesQuimarox".Quimarox[#ID_Quimarox].vagon[#PeineParaReserva].vagon_reservado_carga;

// escribimos el los datos de la entrada el id del elemento que ha realizado la reserva
      L     #ID_ElementoPeticion;
      T     "DB601_PeinesQuimarox".Quimarox[#ID_Quimarox].vagon[#PeineParaReserva].punto_entrada_carga;

      L     #PeineParaReserva;
      T     #NumeroPeineReservado;

      BE;



NETWORK
TITLE = Final >>> Esperar Para Reservar
/////////////////////////////////////////////////////////////////////////////////////
// Si no hemos encontrado ningún carrier libre en el sorter, no podemos
// seguir buscando infinitamente (bucle infinito y el CPU a stop)
// tendremos que lanzar un temporizador de espera para volver a gestionar la busqueda.
EsperaParaReservar:NOP   0;
      BE;


END_FUNCTION

FUNCTION "FC603_ResetQuimarox" : Void   // FC603, LAD
{ S7_Optimized_Access := 'TRUE' }
// stored: AutoNumber false, SetENOAutomatically false
   VAR_INPUT
      ID_Quimarox : UInt;
   END_VAR
   VAR_IN_OUT
      Maux_formateo : Bool;
   END_VAR
   VAR_TEMP
      contador : UInt;
      Mesa_quimarox : UInt;
   END_VAR
BEGIN

NETWORK
TITLE = Distribucion

      L     "DB600_ConfigQuimarox".Quimarox[#ID_Quimarox].datos_config.Numero_MesaAsociada;
      T     #Mesa_quimarox;

      SET;  // No hay que hacer nada
      AN    "DB902_Estado_ZonaMesa".EstadoMesas[#Mesa_quimarox].PerReset_CBx;
      AN    "DB902_Estado_ZonaMesa".EstadoMesas[#Mesa_quimarox].Resetear_CBx;
      JC    fin;

      SET;  // Reseteo --> Enviar eventos
      A     "DB902_Estado_ZonaMesa".EstadoMesas[#Mesa_quimarox].Resetear_CBx;
      AN    #Maux_formateo;
      JC    evento_QRES;

      SET;  // Activar Fin de Reset
      A     "DB902_Estado_ZonaMesa".EstadoMesas[#Mesa_quimarox].PerReset_CBx;
      JC    fin_reset;

      BE;


NETWORK
TITLE = En el proceso de reset, buscamos todos los peines que tengan datos y les escribimos el 503 para envio de mensajes
//==============================================================================================
evento_QRES:NOP   0;


      L     1;
      T     #contador;


bucle:NOP   0;

      SET;
      AN    "DB601_PeinesQuimarox".Quimarox[#ID_Quimarox].vagon[#contador].Carrier_Cargado;
      JC    siguiente;

// como tenemos carga, escribimos el evento que formatea el mensaje del reset

      L     "CTE_Evento_QRST";
      T     "DB601_PeinesQuimarox".Quimarox[#ID_Quimarox].vagon[#contador].EventoAGenerar;

// y pasamos a supervisar el siguiente vagon

//==============================================================================================
siguiente:NOP   0;  // comprobamos si hemos llegado al máximo de los vagones

      L     #contador;
      L     "DB600_ConfigQuimarox".Quimarox[#ID_Quimarox].datos_config.Numero_vagones;
      >=I;
      JC    fin_qres;

// si no hemos saltado es porque nos quedan vagones que revisar

      L     1;
      L     #contador;
      +I;
      T     #contador;

      JU    bucle;

fin_qres:SET;
      S     #Maux_formateo;
      BE;


//==============================================================================================

NETWORK
TITLE = generación del fin de reset
//==============================================================================================
fin_reset:NOP   0;

// para poder dar el fin de reset tenemos que asegurar que todos los mensajes QRES se han enviado

      L     1;
      T     #contador;

bucle2:NOP   0;

      L     "DB601_PeinesQuimarox".Quimarox[#ID_Quimarox].vagon[#contador].EventoAGenerar;
      L     0;
      <>I;
      JC    quedan_mensajes;

// si no hemos saltado es porque nos quedan vagones que revisar

      L     #contador;
      L     "DB600_ConfigQuimarox".Quimarox[#ID_Quimarox].datos_config.Numero_vagones;
      >=I;
      JC    da_fin_reset;


      L     1;
      L     #contador;
      +I;
      T     #contador;

      JU    bucle2;

quedan_mensajes:NOP   0;
      CLR;
      =     "DB900_Estado_Mesas".EstadoVI[#Mesa_quimarox].Fin_VI;
      BE;

da_fin_reset:SET;
      R     #Maux_formateo;
      =     "DB900_Estado_Mesas".EstadoVI[#Mesa_quimarox].Fin_VI;
      BE;


NETWORK
TITLE = 

fin:  SET;
      R     #Maux_formateo;
      =     "DB900_Estado_Mesas".EstadoVI[#Mesa_quimarox].Fin_VI;
      BE;



END_FUNCTION

FUNCTION "FC604_PuntoBorradoDatos_Quimarox" : Void   // FC604, LAD
{ S7_Optimized_Access := 'FALSE' }
// stored: AutoNumber false, SetENOAutomatically false
   VAR_INPUT
      ID_Quimarox : Int;
      ID_Elemento : Int;
   END_VAR
   VAR_TEMP
      Nux_NumeroVagon : Int;
   END_VAR
BEGIN

NETWORK
TITLE = Borrar el Peine del Quimarox
//======================================================================================================================================
// sacamos el dato del vagón que tenemos en frente del elemento:
      L     "DB602_ElementosQuimarox".Quimarox[#ID_Quimarox].Elementos[#ID_Elemento].Numero_carrier;
      T     #Nux_NumeroVagon;

// Numero de Vagon nunca debe ser CERO
      L     #Nux_NumeroVagon;
      L     0;
      ==I;
      JC    fin;

// Hay Carrier en ventana
      SET;
      AN    "DB602_ElementosQuimarox".Quimarox[#ID_Quimarox].Elementos[#ID_Elemento].Hay_Carrier_en_ventana;
      JC    fin;

// primero comprobamos si tenemos algún mensaje pendiente de emitir
      SET;
      L     "DB601_PeinesQuimarox".Quimarox[#ID_Quimarox].vagon[#Nux_NumeroVagon].EventoAGenerar;
      L     0;
      <>I;
      JC    fin;


//========================================================================================================================================
// borramos los datos del vagón, salvo los de la reserva
      SET;
      R     "DB601_PeinesQuimarox".Quimarox[#ID_Quimarox].vagon[#Nux_NumeroVagon].Carrier_Cargado;
      R     "DB601_PeinesQuimarox".Quimarox[#ID_Quimarox].vagon[#Nux_NumeroVagon].vagon_cargado_SinDestino;
      R     "DB601_PeinesQuimarox".Quimarox[#ID_Quimarox].vagon[#Nux_NumeroVagon].carrier_multiple;
//      R     "DB601_DatosPeinesQuimarox".Quimarox[#ID_Quimarox].vagon[#Nux_NumeroVagon].vagon_reservado_carga

      L     0;
      T     "DB601_PeinesQuimarox".Quimarox[#ID_Quimarox].vagon[#Nux_NumeroVagon].Destino_principal;
      T     "DB601_PeinesQuimarox".Quimarox[#ID_Quimarox].vagon[#Nux_NumeroVagon].Destino_alternativo;
      T     "DB601_PeinesQuimarox".Quimarox[#ID_Quimarox].vagon[#Nux_NumeroVagon].Mesa_descarga;
      T     "DB601_PeinesQuimarox".Quimarox[#ID_Quimarox].vagon[#Nux_NumeroVagon].Num_Recirculaciones;
      T     "DB601_PeinesQuimarox".Quimarox[#ID_Quimarox].vagon[#Nux_NumeroVagon].Numero_Vagones_Multiple_Asociados;
//      T     "DB601_DatosPeinesQuimarox".Quimarox[#ID_Quimarox].vagon[#Nux_NumeroVagon].punto_entrada_carga

      L     0;
      T     "DB601_PeinesQuimarox".Quimarox[#ID_Quimarox].vagon[#Nux_NumeroVagon].EventoAGenerar;
      T     "DB601_PeinesQuimarox".Quimarox[#ID_Quimarox].vagon[#Nux_NumeroVagon].DatosCarga.Mckey;
      T     "DB601_PeinesQuimarox".Quimarox[#ID_Quimarox].vagon[#Nux_NumeroVagon].DatosCarga.MesaDestino;
      T     "DB601_PeinesQuimarox".Quimarox[#ID_Quimarox].vagon[#Nux_NumeroVagon].DatosCarga.MesaOrigen;
      T     "DB601_PeinesQuimarox".Quimarox[#ID_Quimarox].vagon[#Nux_NumeroVagon].DatosCarga.EtiquetaRouter;




//========================================================================================================================================
fin:  BE;
END_FUNCTION

FUNCTION "FC608_CambioEstado_Peines" : Void   // FC608, LAD
{ S7_Optimized_Access := 'TRUE' }
// stored: AutoNumber false, SetENOAutomatically false
   VAR_INPUT
      Aplica_Cambio : Bool;
      ID_Quimarox : UInt;
      ID_Peine : UInt;   // Numero_Peine o 999 para ejecutar acción sobre todos los peines
      Acción : UInt;   // 1 Habilitar, 2 Deshabilitar
   END_VAR
   VAR_OUTPUT
      Result : Bool;   // 0 resultado ok, 1 resultado nook
   END_VAR
   VAR_TEMP
      Aux_Contador : UInt;
   END_VAR
BEGIN

NETWORK
TITLE = 0 resultado ok, 1 resultado nook
//======================================================================
// Hasta que no tengamos aplicar cambio, no ejecutamos ninguna acción

      SET;
      AN    #Aplica_Cambio;
      JC    Fin;

//======================================================================
// si la acción es 0, no tenemos que hacer nada

      SET;
      L     #Acción;
      L     0;
      ==I;
      JC    Fin;

//======================================================================
// comprobamos si el ID de quimarox es válido
      SET;
      A(;
      L     #ID_Quimarox;
      L     0;
      <>I;
      );
      A(;
      L     #ID_Quimarox;
      L     "CTE_MaxNumQuimarox";
      <=I;
      );
      JC    rango_quimarox_valido;

//======================================================================
// si el rango no es válido, marcamos result 1 y salimos de la funcióm
      JU    Fin_nok;

//======================================================================
// comprobamos si la acción es sobre un peine o sobre todos
rango_quimarox_valido:NOP   0;

      SET;
      L     #ID_Peine;
      L     999;
      ==I;
      JC    todos_los_peines;

// si la acción no es sobre todos los peines, pasamos a comprobar si el número de peine es válido

      SET;
      A(;
      L     #ID_Peine;
      L     0;
      >I;
      );
      A(;
      L     #ID_Peine;
      L     "DB600_ConfigQuimarox".Quimarox[#ID_Quimarox].datos_config.Numero_vagones;
      <=I;
      );
      JC    rango_peine_valido;
//======================================================================
// si el rango no es válido, marcamos result 1 y salimos de la funcióm

      JU    Fin_nok;

//======================================================================

NETWORK
TITLE = Ejecución de acciones sobre todos los peines
//======================================================================
todos_los_peines:NOP   0;

// inicializamos el contador para movernos por el bucle
      L     1;
      T     #Aux_Contador;

// en función de la acción a ejecutar, vamos a un bucle o a otro
//======================================================================
bucle:L     #Acción;
      JL    LSTX;
      JU    Fin;
      JU    Habilitar_todos;
      JU    Deshabilitar_todos;

LSTX: JU    Fin;
//======================================================================
Habilitar_todos:NOP   0;
      CLR;
      =     "DB601_PeinesQuimarox".Quimarox[#ID_Quimarox].vagon[#Aux_Contador].carrier_no_utilizable;
      JU    Siguiente_Peine;

//======================================================================
Deshabilitar_todos:NOP   0;
      SET;
      =     "DB601_PeinesQuimarox".Quimarox[#ID_Quimarox].vagon[#Aux_Contador].carrier_no_utilizable;
      JU    Siguiente_Peine;
//======================================================================

Siguiente_Peine:NOP   0;
// comprobamos si hemos llegado al final del bucle
      SET;
      L     #Aux_Contador;
      L     "DB600_ConfigQuimarox".Quimarox[#ID_Quimarox].datos_config.Numero_vagones;
      >=I;
      JC    Fin_ok;

// si no hemos acabado, pasamos al siguiente peine

      L     #Aux_Contador;
      L     1;
      +I;
      T     #Aux_Contador;
      JU    bucle;

//======================================================================

NETWORK
TITLE = Ejecución de acciones sobre un peine en concreto
rango_peine_valido:NOP   0;



      L     #Acción;
      JL    LSTXp;
      JU    Fin;
      JU    Habilitar;
      JU    Deshabilitar;

LSTXp:JU    Fin;

//======================================================================
Habilitar:NOP   0;
      CLR;
      =     "DB601_PeinesQuimarox".Quimarox[#ID_Quimarox].vagon[#ID_Peine].carrier_no_utilizable;
      JU    Fin_ok;

//======================================================================
Deshabilitar:NOP   0;
      SET;
      =     "DB601_PeinesQuimarox".Quimarox[#ID_Quimarox].vagon[#ID_Peine].carrier_no_utilizable;
      JU    Fin_ok;
//======================================================================



NETWORK
TITLE = 0 resultado ok, 1 resultado nook
//======================================================================
Fin:  BE;
//======================================================================
Fin_nok:NOP   0;
      SET;
      =     #Result;
      BE;
//======================================================================
Fin_ok:NOP   0;
      CLR;
      =     #Result;
      BE;
//======================================================================
END_FUNCTION

DATA_BLOCK "DB2112_DB_LinPot_2"   // DB2112, F_DB
FAMILY : FPRI0853
VERSION : 0.0
// stored: AutoNumber false, InstanceOfName FB2131_F_Linea_Potencia, InstanceOfType FB
"FB2131_F_Linea_Potencia"
   // VAR_INPUT
   //    NumArmario : Int;
   //    NumLinea : Int;
   //    Desconectar : Bool;
   //    Proteccion : Bool;
   //    Seguridades : Bool;
   //    FEEDBACK : Bool;
   //    ACK_NEC : Bool;
   //    ACK : Bool;
   //    "ACK_ESTA _LINEA" : Bool;
   //    QBAD_FIO : Bool;
   //    FDB_TIME : Time;
   //    TIM_Estabilizacion : Time;
   // END_VAR
   // VAR_OUTPUT
   //    Q : Bool;
   //    ERROR : Bool;
   //    ACK_Next : Bool;
   // END_VAR
   // VAR
   //    F_TON { S7_SetPoint := 'True'} : TON;
   //    F_FDBACK { S7_SetPoint := 'True'} : FDBACK;
   //    F_ESTOP1 { S7_SetPoint := 'True'} : ESTOP1;
   //    Mem_ACK : Bool;
   //    Pos_ACK : Bool;
   // END_VAR
BEGIN
END_DATA_BLOCK

DATA_BLOCK "DB2125_DB_LinPot_Maq1"   // DB2125, F_DB
FAMILY : FPRI0855
VERSION : 0.0
// stored: AutoNumber false, InstanceOfName FB2133_F_LinPot_Maquina, InstanceOfType FB
"FB2133_F_LinPot_Maquina"
   // VAR_INPUT
   //    NumArmario : Int;
   //    NumLinea : Int;
   //    Maquina_OFF : Bool;
   //    Proteccion : Bool;
   //    Seguridades : Bool;
   //    FEEDBACK : Bool;
   //    Rearme : Bool;
   //    QBAD_FIO : Bool;
   //    FDB_TIME : Time;
   // END_VAR
   // VAR_OUTPUT
   //    Q : Bool;
   //    ERROR : Bool;
   //    H : Bool;
   // END_VAR
   // VAR
   //    F_FDBACK { S7_SetPoint := 'True'} : FDBACK;
   //    F_ESTOP1 { S7_SetPoint := 'True'} : ESTOP1;
   // END_VAR
BEGIN
END_DATA_BLOCK

DATA_BLOCK "DB2143_DB_STV1"   // DB2140, F_DB
// stored: AutoNumber false, InstanceOfName FB2143_F_Control_STV, InstanceOfType FB
"FB2143_F_Control_STV"
   // VAR_INPUT
   //    NumArmario : Int;
   //    NumLinea : Int;
   //    Desconectar : Bool;
   //    ACK : Bool;
   //    Setas_OK : Bool;
   //    Error_Protusion : Bool;
   //    Barreras_OK : Bool;
   //    Incendio_OK : Bool;
   //    FeedbackPotencia : Bool;
   //    FeedbackFaseRS : Bool;
   //    QBAD_Potencia : Bool;
   //    QBAD_FaseRS : Bool;
   //    ProteccionPotencia : Bool;
   //    ProteccionFaseRS : Bool;
   //    PuertasSect_Abiertas : Bool;
   //    DFK_FireShutterCloseOK : Bool;
   //    DFK_STV_All_Stop : Bool;
   //    PuertasAcceso_Cerradas : Bool;
   //    Vigilancia_PuertasAcceso : Bool;
   // END_VAR
   // VAR_OUTPUT
   //    DFK_Load_Protrusion : Bool;
   //    DFK_Fire_Alarm : Bool;
   //    DFK_FireShutter_Open : Bool;
   //    Cerrar_Puertas_OK : Bool;
   //    Fases_RS_STV : Bool;
   //    Potencia_STV : Bool;
   //    Error_Potencia : Bool;
   //    Error_FaseRS : Bool;
   //    ACK_Next : Bool;
   // END_VAR
   // VAR
   //    MA_DFK_FireShutter_Open : Bool;
   //    MA_Cerrar_Puertas_OK : Bool;
   //    FB_Potencia_STV { S7_SetPoint := 'True'} : "FB2131_F_Linea_Potencia";
   //    FB_Feedback_FaseRS { S7_SetPoint := 'True'} : FDBACK;
   // END_VAR
BEGIN
END_DATA_BLOCK

DATA_BLOCK "DB1600_DB_CCPIF"   // DB1600
AUTHOR : GENERAL
NAME : 20130301
VERSION : 3.0
// stored: AutoNumber false, InstanceOfName FB900_CONTROL_ZONA, InstanceOfType FB
"FB900_CONTROL_ZONA"
   // VAR_INPUT
   //    NumZonaUP : UInt;
   //    NumZona : UInt;
   //    MAR_FinReset_DW : Bool;
   //    CONF_Reset_Manual : Bool;
   //    INP_Sel_OffLine : Bool;
   //    INP_Sel_Main : Bool;
   //    INP_Pul_Marcha : Bool;
   //    INP_Pul_Paro : Bool;
   //    INP_Pul_Rearme : Bool;
   //    INP_Pul_TLuces : Bool;
   //    INP_Sel_Automat : Bool;
   //    INP_Sel_Manual : Bool;
   // END_VAR
   // VAR_OUTPUT
   //    L_Verde : Bool;
   //    L_Rojo : Bool;
   //    L_Naranja : Bool;
   //    Sirena : Bool;
   // END_VAR
   // VAR
   //    Toff_Rearme { ExternalAccessible := 'False'; ExternalVisible := 'False'; ExternalWritable := 'False'} : TOF_TIME;
   //    TIM_RetardoMarcha { S7_SetPoint := 'True'} : TON_TIME;
   //    Valor_Cuenta_Reset : UDInt;
   //    Modo_Zona_E0 : Bool;
   //    Modo_Zona_E1 : Bool;
   //    Modo_Zona_E2 : Bool;
   //    Modo_Zona_E3 : Bool;
   //    Modo_Zona_E4 : Bool;
   //    Modo_Zona_E5 : Bool;
   //    S_Paro_Zona : Bool;
   //    S_Marcha_Zona : Bool;
   //    Auto_Zona_E0 : Bool;
   //    Auto_Zona_E1 : Bool;
   //    Auto_Zona_E2 : Bool;
   //    Auto_Zona_E3 : Bool;
   //    Auto_Zona_E4 : Bool;
   //    Auto_Zona_E5 : Bool;
   //    Reset_Zona_E0 : Bool;
   //    Reset_Zona_E1 : Bool;
   //    Reset_Zona_E2 : Bool;
   //    Reset_Zona_E3 : Bool;
   //    Reset_Zona_E4 : Bool;
   //    Reset_Zona_E5 : Bool;
   //    Reset_Zona_E6 : Bool;
   //    Reset_Zona_E7 : Bool;
   //    Mem_PulMarcha_Zona : Bool;
   //    Mem_Error_Zona : Bool;
   //    Mem_Aviso_Error_Zona : Bool;
   //    Mem_Parar_Zona : Bool;
   //    Mem_Reseteo_Zona : Bool;
   //    Mem_PulParo_Zona : Bool;
   //    Mem_Fin_Zona : Bool;
   //    Mem_Fin_Reset_Zona : Bool;
   //    Mem_FP_Rearme : Bool;
   //    Mem_Free2 : Bool;
   //    MemoriaSirena : Bool;
   //    Cuenta_Reset_OK : Bool;
   // END_VAR
BEGIN
END_DATA_BLOCK
